Universal Robots PolyScope program: Pour_water.urp

Program Pour_water (installation=default directory=/programs/Matcha createdIn=5.8.2.10297 lastSavedIn=5.12.6.1102099 robotSerialNumber=20215500597)
Calibrated DH parameters: a=[0.000193, -0.066673, -0.391568, -0.000012, 0.00005, 0]; d=[0.162643, -472.05677, 465.132521, 7.058239, 0.099746, 0.099582]; alpha=[1.571116, 0.00089, 0.003862, 1.569269, -1.569248, 0]; deltaTheta=[0, -1.413394, 7.628392, 0.068187, 0, -0.000001]
Robot Program (runOnlyOnce=true)
  MoveJ speed 60 deg/s, acceleration 80 deg/s^2 (useActiveTCP=true) feature=Base
    Waypoint center_1: TCP in base x=-78.584 y=-626.961 z=386.266 mm, rx=0.0115 ry=-2.2034 rz=2.2303 rad; joints [53.978, -98.506, 113.326, -15.858, 53.984, 180.13] deg; TCP offset x=0 y=0 z=191.5 mm, rx=0 ry=0 rz=0 rad
    Waypoint Waypoint_1: TCP in base x=-77.251 y=-679.703 z=322.67 mm, rx=0.0347 ry=-2.8828 rz=1.2266 rad; joints [64.329, -70.997, 66.84, 50.957, 71.587, 160.238] deg
    Wait Sleep waitTime=5
    Waypoint center_1: TCP in base x=-78.584 y=-626.961 z=386.266 mm, rx=0.0115 ry=-2.2034 rz=2.2303 rad; joints [53.978, -98.506, 113.326, -15.858, 53.984, 180.13] deg
